FUNCTION_BLOCK FB_EventLogger
VAR
	aEventBuffer : ARRAY[1..MAXIMUM_SIZE_OF_EVENT_BUFFER] OF ST_Event;
	nCurrentEventBufferIndex : INT := 0; 
END_VAR
VAR CONSTANT
	MAXIMUM_SIZE_OF_EVENT_BUFFER : INT := 100;
END_VAR

(* Returns TRUE if add was successful and FALSE if buffer is full *)
METHOD PUBLIC AddEvent : BOOL
VAR_INPUT
	eEventType : E_EventType;
	eEventSeverity : TcEventSeverity;
	nEventIdentity : UDINT;
	sEventText : STRING(255);
END_VAR
VAR
	stNewEvent : REFERENCE TO ST_Event;
END_VAR
AddEvent := FALSE;

IF IsEventBufferFull() THEN
	RETURN;
END_IF

// Allocate space for a new event in the event buffer
nCurrentEventBufferIndex := nCurrentEventBufferIndex + 1;
stNewEvent REF= aEventBuffer[nCurrentEventBufferIndex];

stNewEvent.eEventType := eEventType;
stNewEvent.eEventSeverity := eEventSeverity;
stNewEvent.nEventIdentity := nEventIdentity;
stNewEvent.sEventText := sEventText;
stNewEvent.dtTimestamp := F_GetSystemDateAndTime();

AddEvent := TRUE;
END_METHOD

METHOD PUBLIC IsEventBufferFull : BOOL
IsEventBufferFull := (nCurrentEventBufferIndex + 1) > MAXIMUM_SIZE_OF_EVENT_BUFFER;
END_METHOD

END_FUNCTION_BLOCK

(* stored: Version 1.1.0.1, ProductVersion 3.1.4024.15
   POU FB_EventLogger: Id {6133763c-6893-4d0d-af70-1ac47f57e8bd}, SpecialFunc None
   Method AddEvent: Id {cad28719-a128-4c96-89b8-26d87b33d667}
   Method IsEventBufferFull: Id {0c1a381c-8331-4785-b133-88efd57b5a7d} *)
